(* Schneider Machine Expert - Basic project prg_control+COUNTER, file version 2.7.0.0 *)
(* ProjectInformations: Name=New project *)

HARDWARE
  Cpu 0: TM221M16R/G
  EthernetConfiguration: NetworkName=M221, IpAllocationMode=FixedAddress, IpAddress=0.0.0.0, SubnetMask=0.0.0.0
  SerialLineConfiguration: Baud=Baud19200, Parity=ParityEven, DataBits=DataBits8, StopBits=StopBits1, PhysicalMedium=PhysicalMediumRs485, TransmissionMode=TransmissionModeModbusRtu, SlaveId=1, Addressing=SlaveAddressing
  MastTask: UsePeriodScanMode=false, PeriodScan=100
  FastTask: Period=255
  CpuBehavior: StartingMode=StartAsPreviousState, AutoSaveRamOnEeprom=true, WatchdogPeriod=250

SYMBOLS  (address, symbol, comment, settings)
  %M0       AUX_MOTOR  "Motor auxilarry"
  %M10      M_START  "M_aux_Start"
  %M11      M_STOP  "M_aux_Stop"
  %M12      M_SENSOR  "M_aux_Sensor"
  %M20      CMD_CONTROL_RESET
  %M21      IND_CONTROL_REACHED
  %M90      IND_ALARM
  %M100     PET_ACK
  %M101     ALARM_01
  %M102     ALARM_02
  %MW0      IND_MOTOR_COUNTER
  %MW11     CFG_COUNTER_MOTOR
  %MW20     IND_MOTOR_TIME
  %MW30     CFG_TIMER_MOTOR
  %TM0      TIMER_MOTOR_ON  [Preset=5, Base=OneSecond]
  %C0         [Preset=5]
  %I0.0     I_START  "start process"
  %I0.1     I_STOP  "stop process"
  %I0.5     I_SENSOR  "detecting"
  %Q0.0     Q_MOTOR  "Motor"
  %Q0.1     Q_MACHINE_ON

POU PRG CONFIG
  (* SectionNumber=1 *)

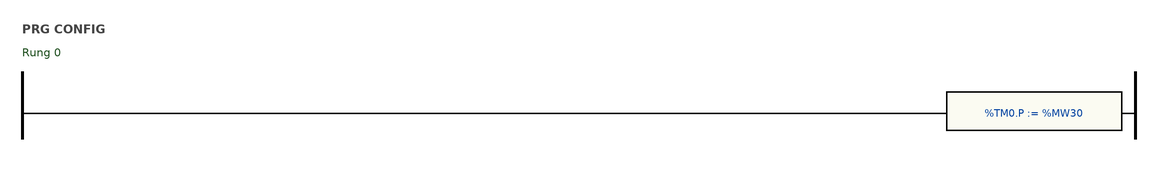

// Rung 0
  LD 1
  [ %TM0.P := %MW30 ]     (* TIMER_MOTOR_ON, CFG_TIMER_MOTOR *)
  // as ST:
  //   TIMER_MOTOR_ON.P := CFG_TIMER_MOTOR;

POU PRG INPUTS
  (* SectionNumber=2 *)

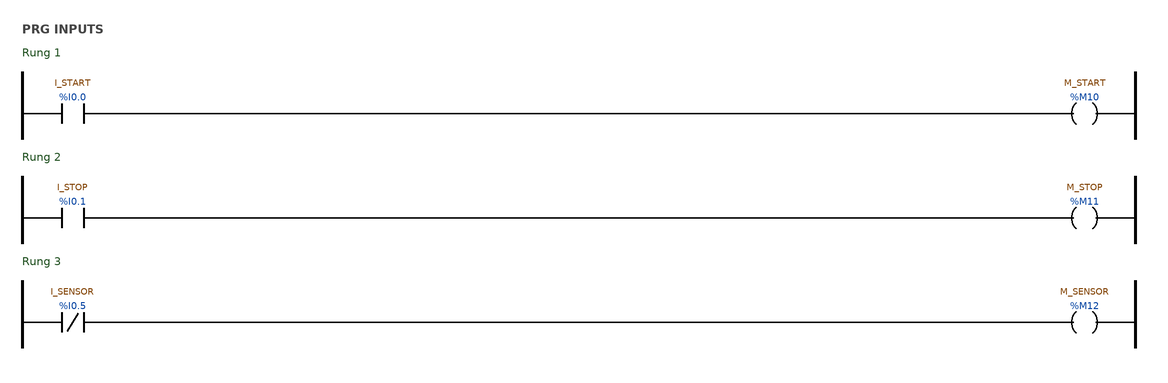

// Rung 1
  LD %I0.0                (* I_START *)
  ST %M10                 (* M_START *)
  // as ST:
  //   M_START := I_START;

// Rung 2
  LD %I0.1                (* I_STOP *)
  ST %M11                 (* M_STOP *)
  // as ST:
  //   M_STOP := I_STOP;

// Rung 3
  LDN %I0.5               (* I_SENSOR *)
  ST %M12                 (* M_SENSOR *)
  // as ST:
  //   M_SENSOR := NOT I_SENSOR;

POU PRG_Control
  (* SectionNumber=3 *)

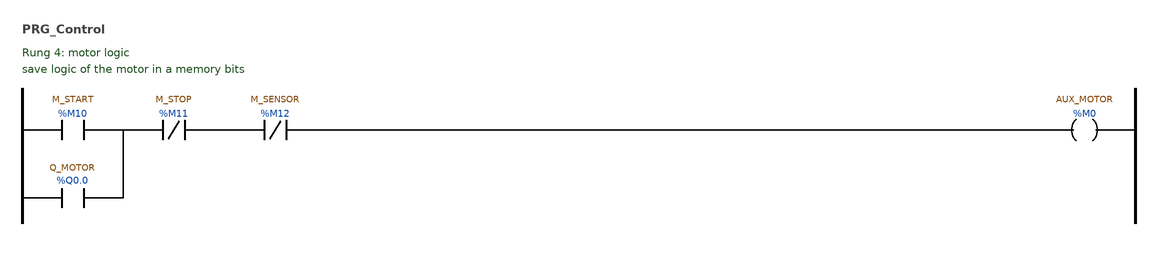

// Rung 4: motor logic
// save logic of the motor in a memory bits
  LD %M10                 (* M_START *)
  OR %Q0.0                (* Q_MOTOR *)
  ANDN %M11               (* M_STOP *)
  ANDN %M12               (* M_SENSOR *)
  ST %M0                  (* AUX_MOTOR *)
  // as ST:
  //   AUX_MOTOR := (M_START OR Q_MOTOR) AND NOT M_STOP AND NOT M_SENSOR;

POU PRG OUTPUT
  (* SectionNumber=4 *)

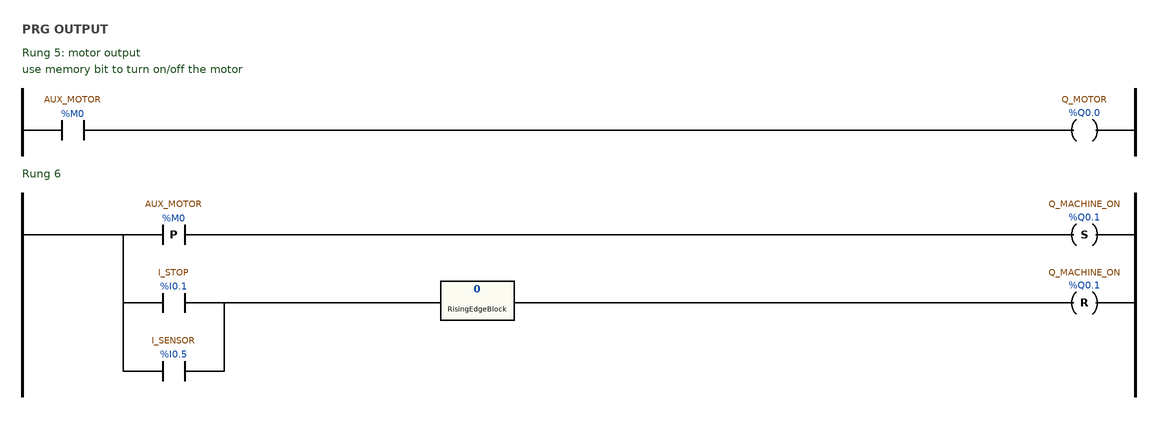

// Rung 5: motor output
// use memory bit to turn on/off the motor
  LD %M0                  (* AUX_MOTOR *)
  ST %Q0.0                (* Q_MOTOR *)
  // as ST:
  //   Q_MOTOR := AUX_MOTOR;

// Rung 6
  LD 1
  MPS
  ANDR %M0                (* AUX_MOTOR *)
  S %Q0.1                 (* Q_MACHINE_ON *)
  MPP
  AND( %I0.1              (* I_STOP *)
  OR %I0.5                (* I_SENSOR *)
  )
  RISING0
  R %Q0.1                 (* Q_MACHINE_ON *)
  // as ST:
  //   IF RISING(AUX_MOTOR) THEN Q_MACHINE_ON := TRUE; END_IF;
  //   IF RISING(I_STOP OR I_SENSOR) THEN Q_MACHINE_ON := FALSE; END_IF;

POU PRG ALArm
  (* SectionNumber=5 *)

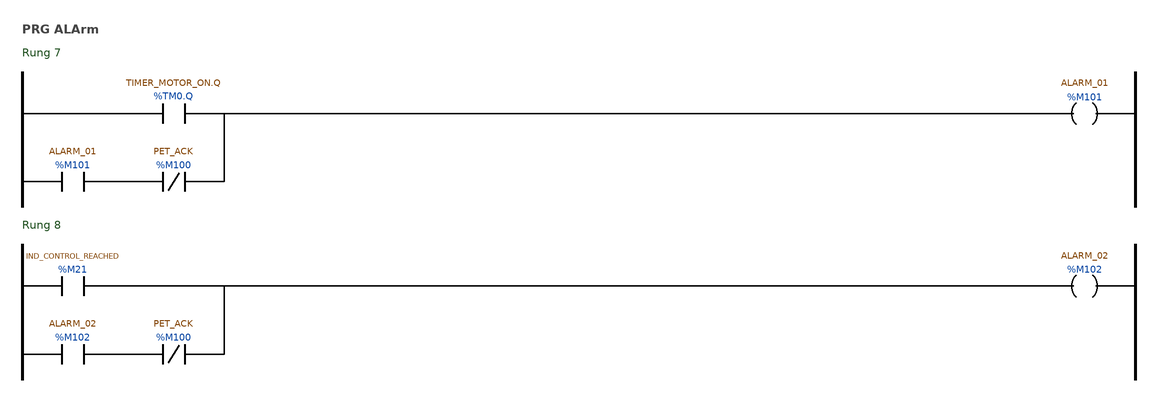

// Rung 7
  LD 1
  AND %TM0.Q              (* TIMER_MOTOR_ON *)
  OR( %M101               (* ALARM_01 *)
  ANDN %M100              (* PET_ACK *)
  )
  ST %M101                (* ALARM_01 *)
  // as ST:
  //   ALARM_01 := TIMER_MOTOR_ON.Q OR ALARM_01 AND NOT PET_ACK;

// Rung 8
  LD %M21                 (* IND_CONTROL_REACHED *)
  OR( %M102               (* ALARM_02 *)
  ANDN %M100              (* PET_ACK *)
  )
  ST %M102                (* ALARM_02 *)
  // as ST:
  //   ALARM_02 := IND_CONTROL_REACHED OR ALARM_02 AND NOT PET_ACK;

POU PRG MGMT
  (* SectionNumber=6 *)

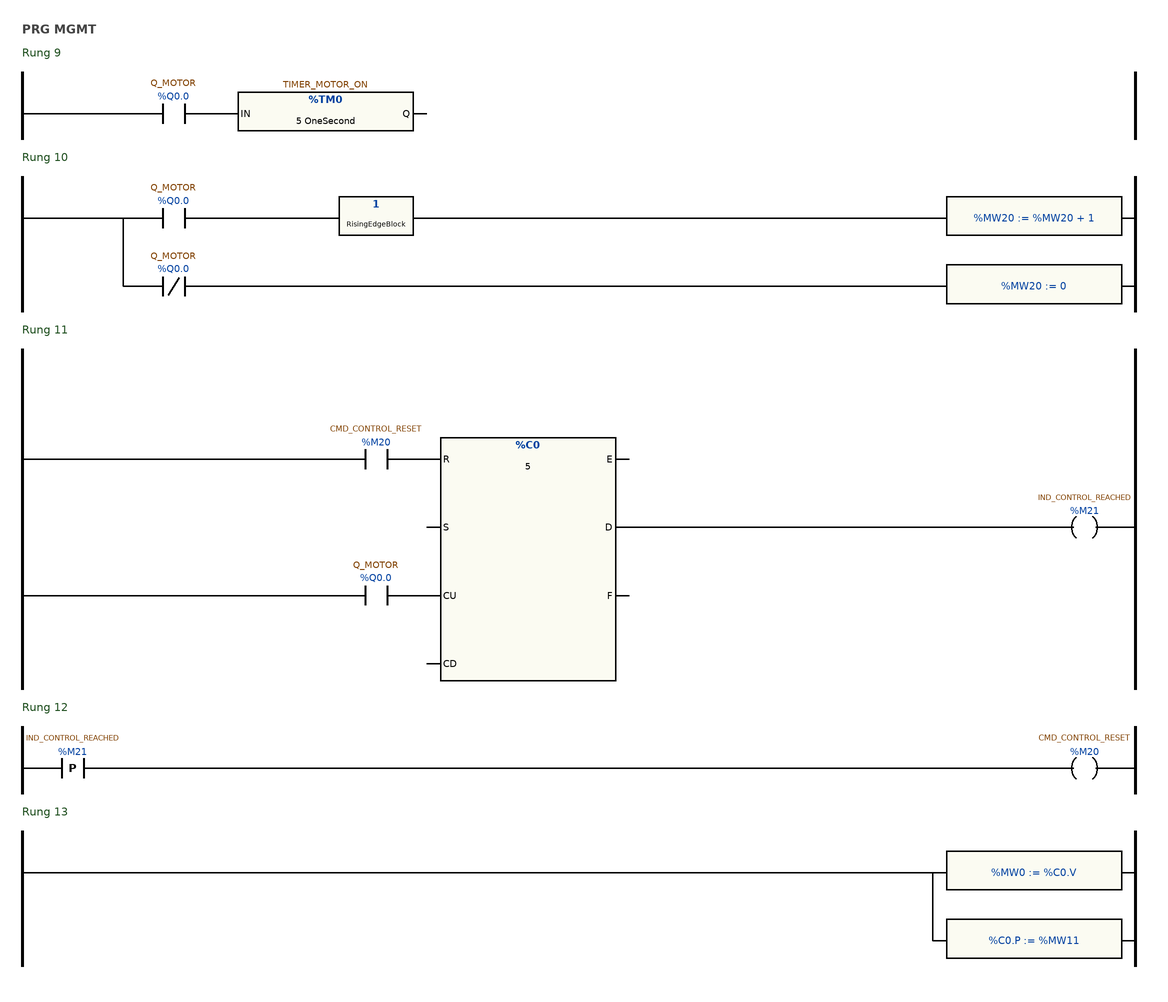

// Rung 9
  BLK %TM0                (* TIMER_MOTOR_ON *)
  LD %Q0.0                (* Q_MOTOR *)
  IN
  END_BLK
  // as ST:
  //   TIMER_MOTOR_ON(IN := Q_MOTOR);

// Rung 10
  LD 1
  MPS
  AND %Q0.0               (* Q_MOTOR *)
  RISING1
  [ %MW20 := %MW20 + 1 ]  (* IND_MOTOR_TIME, IND_MOTOR_TIME *)
  MPP
  ANDN %Q0.0              (* Q_MOTOR *)
  [ %MW20 := 0 ]          (* IND_MOTOR_TIME *)
  // as ST:
  //   IF RISING(Q_MOTOR) THEN IND_MOTOR_TIME := IND_MOTOR_TIME + 1; END_IF;
  //   IF NOT Q_MOTOR THEN IND_MOTOR_TIME := 0; END_IF;

// Rung 11
  BLK %C0
  LD %M20                 (* CMD_CONTROL_RESET *)
  R
  LD %Q0.0                (* Q_MOTOR *)
  CU
  OUT_BLK
  LD D
  ST %M21                 (* IND_CONTROL_REACHED *)
  END_BLK
  // as ST:
  //   %C0(R := CMD_CONTROL_RESET, CU := Q_MOTOR);
  //   IND_CONTROL_REACHED := %C0.D;

// Rung 12
  LDR %M21                (* IND_CONTROL_REACHED *)
  ST %M20                 (* CMD_CONTROL_RESET *)
  // as ST:
  //   CMD_CONTROL_RESET := RISING(IND_CONTROL_REACHED);

// Rung 13
  LD 1
  [ %MW0 := %C0.V ]       (* IND_MOTOR_COUNTER *)
  [ %C0.P := %MW11 ]      (* CFG_COUNTER_MOTOR *)
  // as ST:
  //   IND_MOTOR_COUNTER := %C0.V;
  //   %C0.P := CFG_COUNTER_MOTOR;

POU PRG GRALS ALARM
  (* SectionNumber=0 *)

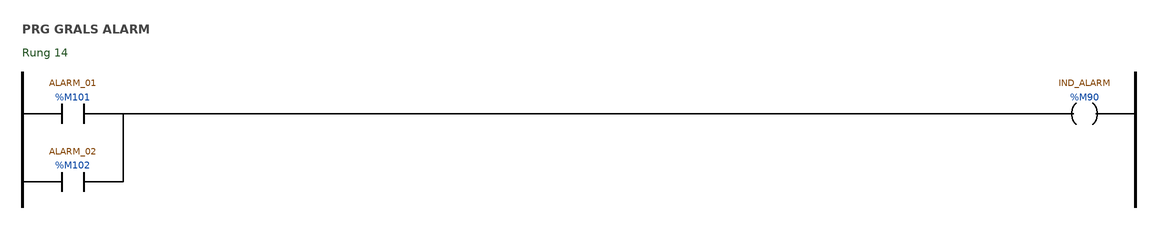

// Rung 14
  LD %M101                (* ALARM_01 *)
  OR %M102                (* ALARM_02 *)
  ST %M90                 (* IND_ALARM *)
  // as ST:
  //   IND_ALARM := ALARM_01 OR ALARM_02;
